// TIA Portal V17 export
// export: Created 2022-01-26T21:47:57.0690455Z, ExportSetting WithDefaults, DisplayName Totally Integrated Automation Portal, DisplayVersion V17, DisplayName TIA Portal Openness, DisplayVersion V17, DisplayName TIA Portal Version Control Interface, DisplayVersion V17, DisplayName STEP 7 Professional, DisplayVersion V17, DisplayName STEP 7 Safety, DisplayVersion V17, DisplayName WinCC Professional, DisplayVersion V17
DATA_BLOCK "InputsSignals"   // DB3
{ S7_Optimized_Access := 'FALSE' }
VERSION : 0.1
// stored: AutoNumber true, DBAccessibleFromOPCUA true, DBAccessibleFromWebserver true, IsOnlyStoredInLoadMemory false, IsWriteProtectedInAS false
   VAR
      iMotor : Bool;
      iManual : Bool;
      iAuto : Bool;
      iSensor : Bool;
      iParo : Bool;
      iVibrador : Bool;
   END_VAR
BEGIN
END_DATA_BLOCK
